FUNCTION_BLOCK ReactorAvCtrl_HMI (* Service Interface Function Block Type *)
  (* Standard: 61499-2 *)
  (* Version 0.0, 7/15/2026, Schneider Electric, template *)
  PACKAGE SE.Nereda;
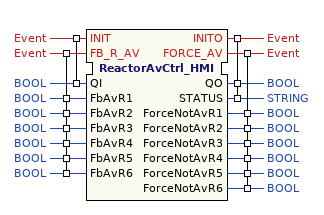
  EVENT_INPUT
    INIT WITH QI;
    FB_R_AV WITH FbAvR1, FbAvR2, FbAvR3, FbAvR4, FbAvR5, FbAvR6;
  END_EVENT
  EVENT_OUTPUT
    INITO WITH QO, STATUS;
    FORCE_AV WITH ForceNotAvR1, ForceNotAvR2, ForceNotAvR3, ForceNotAvR4, ForceNotAvR5, ForceNotAvR6;
  END_EVENT
  VAR_INPUT
    QI : BOOL;
    FbAvR1 : BOOL;
    FbAvR2 : BOOL;
    FbAvR3 : BOOL;
    FbAvR4 : BOOL;
    FbAvR5 : BOOL;
    FbAvR6 : BOOL;
  END_VAR
  VAR_OUTPUT
    QO : BOOL; (* Event Output Qualifier *)
    STATUS : STRING; (* Service Status *)
    ForceNotAvR1 : BOOL;
    ForceNotAvR2 : BOOL;
    ForceNotAvR3 : BOOL;
    ForceNotAvR4 : BOOL;
    ForceNotAvR5 : BOOL;
    ForceNotAvR6 : BOOL;
  END_VAR
  SERVICE /
    SEQUENCE 
    END_SEQUENCE
  END_SERVICE
END_FUNCTION_BLOCK
